               IF (gtyp_SSC.Horizontal_Axis.di_Actual_Position <= (ldi_Pos_Horizontal + gtyp_SSC.Horizontal_Axis.Config.di_Pos_Window))
                   AND (gtyp_SSC.Horizontal_Axis.di_Actual_Position >= (ldi_Pos_Horizontal - gtyp_SSC.Horizontal_Axis.Config.di_Pos_Window))
                   AND gtyp_SSC.Horizontal_Axis.x_Position_Reached
                   AND (gtyp_SSC.Vertical_Axis.di_Actual_Position <= (ldi_Pos_Vertical + gtyp_SSC.Vertical_Axis.Config.di_Pos_Window))
                   AND (gtyp_SSC.Vertical_Axis.di_Actual_Position >= (ldi_Pos_Vertical - gtyp_SSC.Vertical_Axis.Config.di_Pos_Window))
                   AND gtyp_SSC.Vertical_Axis.x_Position_Reached THEN
                   gtyp_SSC.Horizontal_Axis.x_Start_Positioning := FALSE;
                   gtyp_SSC.Vertical_Axis.x_Start_Positioning := FALSE;
                   gtyp_Setup.x_Start_Positioning := FALSE;
                   li_StepCase := 60;
               END_IF;

           60:


               IF gtyp_Setup.x_Start_Positioning OR gtyp_Setup.x_Home_Positioning THEN
                   lx_Start_Positioning_m := TRUE;
                   li_StepCase            := 10;
               ELSIF lfb_R_Trig_Deaktivate.Q THEN
                   gtyp_Setup.x_Home_Positioning := FALSE;
                   li_StepCase                    := 70;
               END_IF;

           70:

               gtyp_SSC.Horizontal_Axis.x_Reference := TRUE;
               gtyp_SSC.Vertical_Axis.x_Reference := TRUE;

               IF NOT gtyp_SSC.Horizontal_Axis.x_Referenced AND NOT gtyp_SSC.Vertical_Axis.x_Referenced THEN
                   li_StepCase := 80;
               END_IF;

           80:
               IF gtyp_SSC.Horizontal_Axis.x_Referenced THEN
                   gtyp_SSC.Horizontal_Axis.x_Reference := FALSE;
               END_IF;
               IF gtyp_SSC.Vertical_Axis.x_Referenced THEN
                   gtyp_SSC.Vertical_Axis.x_Reference := FALSE;
               END_IF;

               IF gtyp_SSC.Horizontal_Axis.x_Referenced AND gtyp_SSC.Vertical_Axis.x_Referenced THEN
                   gtyp_SSC.Horizontal_Axis.x_Reference := FALSE;
                   gtyp_SSC.Vertical_Axis.x_Reference := FALSE;
                   li_StepCase := 0;
               END_IF;


           ELSE
               ;
       END_CASE;

       IF ((gtyp_Setup.i_Pos_Selection > 0)
           AND (gtyp_Setup.i_Pos_Selection < 21)) THEN

           gtyp_Setup.di_Pos_Horizontal := ldi_Pos_Horizontal;
           gtyp_Setup.di_Pos_Vertical := ldi_Pos_Vertical;
           gtyp_Setup.di_Pos_Rotate := 0;
       END_IF;
   ELSE
       lx_Init := TRUE;
   END_IF;
END_FUNCTION_BLOCK

FUNCTION_BLOCK PRG_HBW_Set_Positioning
   VAR
      lx_Init : Bool;
      lx_Start_TON_Wait : Bool;
      lx_Start_Positioning_m : Bool;
      lx_Start_FinalPositioning_m : Bool;
      lx_Start_Offset_m : Bool;
      lt_TON_Wait : Time;
      li_Counter_Hor : Int;
      li_Counter_Ver : Int;
      li_Counter_Act_Hor : Int;
      li_Counter_Act_Ver : Int;
      li_Counter : Int;
      li_StepCase : Int;
      ldi_Pos_Horizontal : DInt;
      ldi_Pos_Vertical : DInt;
      ldi_Offset_Vertical : DInt;
      lfb_R_Trig_Deaktivate : R_TRIG;
      lfb_TON_Wait : TON_TIME;
   END_VAR



   IF lx_Init THEN


       lfb_TON_Wait(IN := lx_Start_TON_Wait,
                     PT := lt_TON_Wait);

       lfb_R_Trig_Deaktivate(CLK:= NOT gtyp_Setup.x_Set_Pos_Activ
                              OR NOT ((gtyp_Setup.i_Pos_Selection > 20)
                              AND (gtyp_Setup.i_Pos_Selection < 41)));

       IF lfb_R_Trig_Deaktivate.Q THEN
           gtyp_HBW.Horizontal_Axis.x_Start_Positioning := FALSE;
           gtyp_HBW.Vertical_Axis.x_Start_Positioning := FALSE;
           gtyp_HBW.Horizontal_Axis.x_Reference := FALSE;
           gtyp_HBW.Vertical_Axis.x_Reference := FALSE;
           gtyp_Setup.x_Start_Positioning := FALSE;
           gtyp_Setup.x_Final_Positioning := FALSE;
           gtyp_Setup.x_Home_Positioning := FALSE;
           gtyp_Setup.x_Start_Offset := FALSE;
           QX_HBW_M4_CantileverBackward_Q8 := FALSE;
           QX_HBW_M4_CantileverForward_Q7 := FALSE;
           IF (li_StepCase > 10) THEN
               li_StepCase := 110;
           END_IF;
       END_IF;


       IF gtyp_Setup.x_Set_Pos_Activ
           AND ((gtyp_Setup.i_Pos_Selection > 20)
           AND (gtyp_Setup.i_Pos_Selection < 41))
           AND ((li_StepCase = 40)
           OR (li_StepCase = 60)
           OR (li_StepCase = 80)
           OR (li_StepCase = 100)) THEN



           IF gtyp_Setup.i_Pos_Selection = 21 THEN
               ldi_Pos_Horizontal := gtyp_HBW.di_PosBelt_Horizontal;
               ldi_Pos_Vertical := gtyp_HBW.di_PosBelt_Vertical;
               ldi_Offset_Vertical := gtyp_HBW.di_Offset_Pos_Belt_Vertical;

           ELSIF gtyp_Setup.i_Pos_Selection = 22 THEN
               ldi_Pos_Horizontal := gtyp_HBW.di_PosRack_A1_Horizontal;
               ldi_Pos_Vertical := gtyp_HBW.di_PosRack_A1_Vertical;
               ldi_Offset_Vertical := gtyp_HBW.di_Offset_Pos_Rack_Vertical;

           ELSIF gtyp_Setup.i_Pos_Selection = 23 THEN
               ldi_Pos_Horizontal := gtyp_HBW.di_PosRack_B2_Horizontal;
               ldi_Pos_Vertical := gtyp_HBW.di_PosRack_B2_Vertical;
               ldi_Offset_Vertical := gtyp_HBW.di_Offset_Pos_Rack_Vertical;

           ELSIF gtyp_Setup.i_Pos_Selection = 24 THEN
               ldi_Pos_Horizontal := gtyp_HBW.di_PosRack_C3_Horizontal;
               ldi_Pos_Vertical := gtyp_HBW.di_PosRack_C3_Vertical;
               ldi_Offset_Vertical := gtyp_HBW.di_Offset_Pos_Rack_Vertical;
           END_IF;
       END_IF;


       IF NOT gtyp_Setup.x_Set_Pos_Activ THEN
           gtyp_Setup.i_Pos_Selection := 0;
       END_IF;


       CASE li_StepCase OF

           0:
               lx_Start_TON_Wait := FALSE;
               li_StepCase := 10;

           10:
               IF gtyp_Setup.x_Set_Pos_Activ
                   AND ((gtyp_Setup.i_Pos_Selection > 20)
                   AND (gtyp_Setup.i_Pos_Selection < 41)) THEN

                   gtyp_HBW.Horizontal_Axis.x_Start_Positioning  := FALSE;
                   gtyp_HBW.Vertical_Axis.x_Start_Positioning    := FALSE;
                   gtyp_HBW.Horizontal_Axis.x_Reference          := FALSE;
                   gtyp_HBW.Vertical_Axis.x_Reference            := FALSE;
                   gtyp_Setup.x_Start_Positioning            := FALSE;
                   gtyp_Setup.x_Final_Positioning            := FALSE;
                   gtyp_Setup.x_Home_Positioning             := FALSE;
                   gtyp_Setup.x_Start_Offset                 := FALSE;
                   QX_HBW_M4_CantileverBackward_Q8               := FALSE;
                   QX_HBW_M4_CantileverForward_Q7                := FALSE;
                   li_StepCase                                    := 20;
               END_IF;

           20:

               gtyp_HBW.Horizontal_Axis.x_Reference := TRUE;
               gtyp_HBW.Vertical_Axis.x_Reference := TRUE;

               IF NOT gtyp_HBW.Horizontal_Axis.x_Referenced AND NOT gtyp_HBW.Vertical_Axis.x_Referenced THEN
                   li_StepCase := 30;
               END_IF;

           30:
               IF gtyp_HBW.Horizontal_Axis.x_Referenced THEN
                   gtyp_HBW.Horizontal_Axis.x_Reference := FALSE;
               END_IF;
               IF gtyp_HBW.Vertical_Axis.x_Referenced THEN
                   gtyp_HBW.Vertical_Axis.x_Reference := FALSE;
               END_IF;

               IF gtyp_HBW.Horizontal_Axis.x_Referenced AND gtyp_HBW.Vertical_Axis.x_Referenced THEN
                   gtyp_HBW.Horizontal_Axis.x_Reference := FALSE;
                   gtyp_HBW.Vertical_Axis.x_Reference := FALSE;
                   li_StepCase := 40;
               END_IF;

           40:
               IF gtyp_Setup.x_Start_Positioning OR lx_Start_Positioning_m OR lx_Start_FinalPositioning_m OR lx_Start_Offset_m THEN
                   lx_Start_Positioning_m := FALSE;
                   li_StepCase := 50;
               END_IF;

           50:
               gtyp_HBW.Horizontal_Axis.di_Target_Position   := ldi_Pos_Horizontal;
               gtyp_HBW.Horizontal_Axis.x_Start_Positioning  := TRUE;
               gtyp_HBW.Vertical_Axis.di_Target_Position     := ldi_Pos_Vertical;
               gtyp_HBW.Vertical_Axis.x_Start_Positioning    := TRUE;

               IF (gtyp_HBW.Horizontal_Axis.di_Actual_Position <= (ldi_Pos_Horizontal + gtyp_HBW.Horizontal_Axis.Config.di_Pos_Window))
                   AND (gtyp_HBW.Horizontal_Axis.di_Actual_Position >= (ldi_Pos_Horizontal - gtyp_HBW.Horizontal_Axis.Config.di_Pos_Window))
                   AND gtyp_HBW.Horizontal_Axis.x_Position_Reached THEN
                   gtyp_HBW.Horizontal_Axis.x_Start_Positioning := FALSE;
               END_IF;

               IF (gtyp_HBW.Vertical_Axis.di_Actual_Position <= (ldi_Pos_Vertical + gtyp_HBW.Vertical_Axis.Config.di_Pos_Window))
                   AND (gtyp_HBW.Vertical_Axis.di_Actual_Position >= (ldi_Pos_Vertical - gtyp_HBW.Vertical_Axis.Config.di_Pos_Window))
                   AND gtyp_HBW.Vertical_Axis.x_Position_Reached THEN
                   gtyp_HBW.Vertical_Axis.x_Start_Positioning := FALSE;
               END_IF;

               IF (gtyp_HBW.Horizontal_Axis.di_Actual_Position <= (ldi_Pos_Horizontal + gtyp_HBW.Horizontal_Axis.Config.di_Pos_Window))
                   AND (gtyp_HBW.Horizontal_Axis.di_Actual_Position >= (ldi_Pos_Horizontal - gtyp_HBW.Horizontal_Axis.Config.di_Pos_Window))
                   AND gtyp_HBW.Horizontal_Axis.x_Position_Reached
                   AND (gtyp_HBW.Vertical_Axis.di_Actual_Position <= (ldi_Pos_Vertical + gtyp_HBW.Vertical_Axis.Config.di_Pos_Window))
                   AND (gtyp_HBW.Vertical_Axis.di_Actual_Position >= (ldi_Pos_Vertical - gtyp_HBW.Vertical_Axis.Config.di_Pos_Window))
                   AND gtyp_HBW.Vertical_Axis.x_Position_Reached THEN
                   gtyp_HBW.Horizontal_Axis.x_Start_Positioning  := FALSE;
                   gtyp_HBW.Vertical_Axis.x_Start_Positioning    := FALSE;
                   gtyp_Setup.x_Start_Positioning          := FALSE;
                   li_StepCase := 60;
               END_IF;

           60:


               IF gtyp_Setup.x_Start_Positioning THEN
                   lx_Start_Positioning_m := TRUE;
                   li_StepCase := 10;

               ELSIF gtyp_Setup.x_Final_Positioning OR lx_Start_FinalPositioning_m OR lx_Start_Offset_m THEN
                   lx_Start_FinalPositioning_m := FALSE;
                   li_StepCase := 70;

               ELSIF lfb_R_Trig_Deaktivate.Q OR gtyp_Setup.x_Home_Positioning THEN
                   gtyp_Setup.x_Home_Positioning := FALSE;
                   li_StepCase := 110;
               END_IF;

           70:

               QX_HBW_M4_CantileverBackward_Q8 := FALSE;
               QX_HBW_M4_CantileverForward_Q7 := TRUE;

               IF IX_HBW_SwitchCantileverFront_I5 AND NOT IX_HBW_SwitchCantileverBack_I6 THEN
                   QX_HBW_M4_CantileverBackward_Q8 := FALSE;
                   QX_HBW_M4_CantileverForward_Q7 := FALSE;
                   gtyp_Setup.x_Final_Positioning := FALSE;
                   li_StepCase := 80;
               END_IF;

           80:


               IF gtyp_Setup.x_Start_Positioning THEN
                   lx_Start_Positioning_m := TRUE;
                   li_StepCase := 110;

               ELSIF gtyp_Setup.x_Final_Positioning THEN
                   lx_Start_FinalPositioning_m := TRUE;
                   li_StepCase := 110;

               ELSIF gtyp_Setup.x_Start_Offset OR lx_Start_Offset_m THEN
                   lx_Start_Offset_m := FALSE;
                   li_StepCase := 90;

               ELSIF lfb_R_Trig_Deaktivate.Q OR gtyp_Setup.x_Home_Positioning THEN
                   gtyp_Setup.x_Home_Positioning := FALSE;
                   li_StepCase := 110;
               END_IF;

           90:
               gtyp_HBW.Vertical_Axis.di_Target_Position := ldi_Pos_Vertical - ldi_Offset_Vertical;
               gtyp_HBW.Vertical_Axis.x_Start_Positioning := TRUE;

               IF (gtyp_HBW.Vertical_Axis.di_Actual_Position <= (ldi_Pos_Vertical - ldi_Offset_Vertical + gtyp_HBW.Vertical_Axis.Config.di_Pos_Window))
                   AND (gtyp_HBW.Vertical_Axis.di_Actual_Position >= (ldi_Pos_Vertical - ldi_Offset_Vertical - gtyp_HBW.Vertical_Axis.Config.di_Pos_Window))
                   AND gtyp_HBW.Vertical_Axis.x_Position_Reached THEN
                   gtyp_HBW.Vertical_Axis.x_Start_Positioning := FALSE;
                   gtyp_Setup.x_Start_Offset            := FALSE;
                   li_StepCase := 100;
               END_IF;

           100:


               IF gtyp_Setup.x_Start_Positioning THEN
                   lx_Start_Positioning_m := TRUE;
                   li_StepCase := 110;

               ELSIF gtyp_Setup.x_Final_Positioning THEN
                   lx_Start_FinalPositioning_m := TRUE;
                   li_StepCase := 110;

               ELSIF gtyp_Setup.x_Start_Offset THEN
                   lx_Start_Offset_m := true;
                   li_StepCase := 110;

               ELSIF lfb_R_Trig_Deaktivate.Q OR gtyp_Setup.x_Home_Positioning THEN
                   gtyp_Setup.x_Home_Positioning := FALSE;
                   li_StepCase := 110;
               END_IF;

           110:
               gtyp_HBW.Vertical_Axis.di_Target_Position := ldi_Pos_Vertical;
               gtyp_HBW.Vertical_Axis.x_Start_Positioning := TRUE;

               IF (gtyp_HBW.Vertical_Axis.di_Actual_Position <= (ldi_Pos_Vertical + gtyp_HBW.Vertical_Axis.Config.di_Pos_Window))
                   AND (gtyp_HBW.Vertical_Axis.di_Actual_Position >= (ldi_Pos_Vertical - gtyp_HBW.Vertical_Axis.Config.di_Pos_Window))
                   AND gtyp_HBW.Vertical_Axis.x_Position_Reached THEN
                   gtyp_HBW.Vertical_Axis.x_Start_Positioning := FALSE;
                   li_StepCase := 120;
               END_IF;

           120:

               QX_HBW_M4_CantileverBackward_Q8 := TRUE;
               QX_HBW_M4_CantileverForward_Q7 := FALSE;

               IF NOT IX_HBW_SwitchCantileverFront_I5 AND IX_HBW_SwitchCantileverBack_I6 THEN
                   QX_HBW_M4_CantileverBackward_Q8 := FALSE;
                   QX_HBW_M4_CantileverForward_Q7 := FALSE;
                   li_StepCase := 130;
               END_IF;

           130:

               gtyp_HBW.Horizontal_Axis.x_Reference := TRUE;
               gtyp_HBW.Vertical_Axis.x_Reference := TRUE;

               IF NOT gtyp_HBW.Horizontal_Axis.x_Referenced AND NOT gtyp_HBW.Vertical_Axis.x_Referenced THEN
                   li_StepCase := 140;
               END_IF;

           140:
               IF gtyp_HBW.Horizontal_Axis.x_Referenced THEN
                   gtyp_HBW.Horizontal_Axis.x_Reference := FALSE;
               END_IF;
               IF gtyp_HBW.Vertical_Axis.x_Referenced THEN
                   gtyp_HBW.Vertical_Axis.x_Reference := FALSE;
               END_IF;

               IF gtyp_HBW.Horizontal_Axis.x_Referenced AND gtyp_HBW.Vertical_Axis.x_Referenced THEN
                   gtyp_HBW.Horizontal_Axis.x_Reference := FALSE;
                   gtyp_HBW.Vertical_Axis.x_Reference := FALSE;
                   li_StepCase := 0;
               END_IF;


       ELSE
           ;
       END_CASE;

       IF ((gtyp_Setup.i_Pos_Selection > 20)
           AND (gtyp_Setup.i_Pos_Selection < 41)) THEN

           gtyp_Setup.di_Pos_Horizontal := ldi_Pos_Horizontal;
           gtyp_Setup.di_Pos_Vertical := ldi_Pos_Vertical;
           gtyp_Setup.di_Pos_Rotate := 0;
       END_IF;
   ELSE
       lx_Init := TRUE;
   END_IF;
END_FUNCTION_BLOCK

FUNCTION_BLOCK PRG_VGR_Set_Positioning
   VAR
      lx_Init : Bool;
      lx_Start_TON_Wait : Bool;
      lx_Start_Positioning_m : Bool;
      lx_Start_FinalPositioning_m : Bool;
      lx_Start_TON_State : Bool;
      lt_TON_Wait : Time;
      ldt_MQTT : Date_And_Time;
      li_Return_LDT : Int;
      li_Lights : Int;
      li_Lights_old : Int;
      lx_State_activ : Bool;
      li_StepCase : Int;
      li_Counter : Int;
      ldi_Pos_SLD_X : DInt;
      ldi_Pos_SLD_Y : DInt;
      ldi_Pos_SLD_Z : DInt;
      ldi_Pos_Horizontal : DInt;
      ldi_Pos_Vertical : DInt;
      ldi_Pos_Rotate : DInt;
      ldi_Offset_Vertical : DInt;
      ls_Color : String;
      ls_Target : String;
      lfb_TON_Wait : TON_TIME;
      lfb_TON_State : TON_TIME;
      lfb_R_Trig_Deaktivate : R_TRIG;
      lfb_R_Trig_NiO : R_TRIG;
   END_VAR



   IF lx_Init THEN


       lfb_TON_Wait(IN := lx_Start_TON_Wait,
                     PT := lt_TON_Wait);

       lfb_R_Trig_Deaktivate(CLK := NOT gtyp_Setup.x_Set_Pos_Activ
                              OR NOT ((gtyp_Setup.i_Pos_Selection > 40)
                              AND (gtyp_Setup.i_Pos_Selection < 61)));

       IF lfb_R_Trig_Deaktivate.Q THEN
           gtyp_VGR.horizontal_Axis.x_Start_Positioning := FALSE;
           gtyp_VGR.vertical_Axis.x_Start_Positioning := FALSE;
           gtyp_VGR.rotate_Axis.x_Start_Positioning := FALSE;
           gtyp_VGR.horizontal_Axis.x_Reference := FALSE;
           gtyp_VGR.vertical_Axis.x_Reference := FALSE;
           gtyp_VGR.rotate_Axis.x_Reference := FALSE;
           gtyp_Setup.x_Start_Positioning := FALSE;
           gtyp_Setup.x_Final_Positioning := FALSE;
           gtyp_Setup.x_Home_Positioning := FALSE;
           gtyp_Setup.x_Start_Offset := FALSE;
           IF (li_StepCase > 10) THEN
               li_StepCase := 150;
           END_IF;
       END_IF;


       IF gtyp_Setup.x_Set_Pos_Activ
           AND ((gtyp_Setup.i_Pos_Selection > 40)
           AND (gtyp_Setup.i_Pos_Selection < 61))
           AND ((li_StepCase = 80)
           OR (li_StepCase = 120)
           OR (li_StepCase = 140)) THEN



           IF gtyp_Setup.i_Pos_Selection = 41 THEN
               ldi_Pos_Horizontal := gtyp_VGR.di_Pos_Color_horizontal;
               ldi_Pos_Vertical := gtyp_VGR.di_Pos_Color_vertical;
               ldi_Pos_Rotate := gtyp_VGR.di_Pos_Color_rotate;
               ldi_Offset_Vertical := gtyp_VGR.di_Offset_Pos_DSI_NFC_vertical;

           ELSIF gtyp_Setup.i_Pos_Selection = 42 THEN
               ldi_Pos_Horizontal := gtyp_VGR.di_Pos_DSI_horizontal;
               ldi_Pos_Vertical := gtyp_VGR.di_Pos_DSI_Collect_vertical;
               ldi_Pos_Rotate := gtyp_VGR.di_Pos_DSI_rotate;
               ldi_Offset_Vertical := gtyp_VGR.di_Offset_Pos_DSI_NFC_vertical;

           ELSIF gtyp_Setup.i_Pos_Selection = 43 THEN
               ldi_Pos_Horizontal := gtyp_VGR.di_Pos_DSI_horizontal;
               ldi_Pos_Vertical := gtyp_VGR.di_Pos_DSI_Discard_vertical;
               ldi_Pos_Rotate := gtyp_VGR.di_Pos_DSI_rotate;
               ldi_Offset_Vertical := gtyp_VGR.di_Offset_Pos_DSI_NFC_vertical;

           ELSIF gtyp_Setup.i_Pos_Selection = 44 THEN
               ldi_Pos_Horizontal := gtyp_VGR.di_Pos_DSO_horizontal;
               ldi_Pos_Vertical := gtyp_VGR.di_Pos_DSO_Collect_vertical;
               ldi_Pos_Rotate := gtyp_VGR.di_Pos_DSO_rotate;
               ldi_Offset_Vertical := gtyp_VGR.di_Offset_Pos_DSO_vertical;

           ELSIF gtyp_Setup.i_Pos_Selection = 45 THEN
               ldi_Pos_Horizontal := gtyp_VGR.di_Pos_DSO_horizontal;
               ldi_Pos_Vertical := gtyp_VGR.di_Pos_DSO_Discard_vertical;
               ldi_Pos_Rotate := gtyp_VGR.di_Pos_DSO_rotate;
               ldi_Offset_Vertical := gtyp_VGR.di_Offset_Pos_DSO_vertical;

           ELSIF gtyp_Setup.i_Pos_Selection = 46 THEN
               ldi_Pos_Horizontal := gtyp_VGR.di_Pos_HBW_horizontal;
               ldi_Pos_Vertical := gtyp_VGR.di_Pos_HBW_Collect_vertical;
               ldi_Pos_Rotate := gtyp_VGR.di_Pos_HBW_rotate;
               ldi_Offset_Vertical := gtyp_VGR.di_Offset_Pos_HBW_vertical;

           ELSIF gtyp_Setup.i_Pos_Selection = 47 THEN
               ldi_Pos_Horizontal := gtyp_VGR.di_Pos_HBW_horizontal;
               ldi_Pos_Vertical := gtyp_VGR.di_Pos_HBW_Discard_vertical;
               ldi_Pos_Rotate := gtyp_VGR.di_Pos_HBW_rotate;
               ldi_Offset_Vertical := gtyp_VGR.di_Offset_Pos_HBW_vertical;

           ELSIF gtyp_Setup.i_Pos_Selection = 48 THEN
               ldi_Pos_Horizontal := gtyp_VGR.di_Pos_MPO_horizontal;
               ldi_Pos_Vertical := gtyp_VGR.di_Pos_MPO_vertical;
               ldi_Pos_Rotate := gtyp_VGR.di_Pos_MPO_rotate;
               ldi_Offset_Vertical := gtyp_VGR.di_Offset_Pos_MPO_vertical;

           ELSIF gtyp_Setup.i_Pos_Selection = 49 THEN
               ldi_Pos_Horizontal := gtyp_VGR.di_Pos_NFC_horizontal;
               ldi_Pos_Vertical := gtyp_VGR.di_Pos_NFC_vertical;
               ldi_Pos_Rotate := gtyp_VGR.di_Pos_NFC_rotate;
               ldi_Offset_Vertical := gtyp_VGR.di_Offset_Pos_DSI_NFC_vertical;

           ELSIF gtyp_Setup.i_Pos_Selection = 50 THEN
               ldi_Pos_Horizontal := gtyp_VGR.di_Pos_NiO_horizontal;
               ldi_Pos_Vertical := gtyp_VGR.di_Pos_NiO_vertical;
               ldi_Pos_Rotate := gtyp_VGR.di_Pos_NiO_rotate;
               ldi_Offset_Vertical := 500;

           ELSIF gtyp_Setup.i_Pos_Selection = 51 THEN
               ldi_Pos_Horizontal := gtyp_VGR.di_Pos_SLD_Blue_horizontal;
               ldi_Pos_Vertical := gtyp_VGR.di_Pos_SLD_Blue_vertical;
               ldi_Pos_Rotate := gtyp_VGR.di_Pos_SLD_Blue_rotate;
               ldi_Offset_Vertical := 500;

           ELSIF gtyp_Setup.i_Pos_Selection = 52 THEN
               ldi_Pos_Horizontal := gtyp_VGR.di_Pos_SLD_Red_horizontal;
               ldi_Pos_Vertical := gtyp_VGR.di_Pos_SLD_Red_vertical;
               ldi_Pos_Rotate := gtyp_VGR.di_Pos_SLD_Red_rotate;
               ldi_Offset_Vertical := 500;

           ELSIF gtyp_Setup.i_Pos_Selection = 53 THEN
               ldi_Pos_Horizontal := gtyp_VGR.di_Pos_SLD_White_horizontal;
               ldi_Pos_Vertical := gtyp_VGR.di_Pos_SLD_White_vertical;
               ldi_Pos_Rotate := gtyp_VGR.di_Pos_SLD_White_rotate;
               ldi_Offset_Vertical := 500;
           END_IF;
       END_IF;


       IF NOT gtyp_Setup.x_Set_Pos_Activ THEN
           gtyp_Setup.i_Pos_Selection := 0;
       END_IF;


       CASE li_StepCase OF

           0:
               lx_Start_TON_Wait := FALSE;
               li_StepCase := 10;

           10:
               IF gtyp_Setup.x_Set_Pos_Activ
                   AND ((gtyp_Setup.i_Pos_Selection > 40)
                   AND (gtyp_Setup.i_Pos_Selection < 61)) THEN

                   gtyp_VGR.horizontal_Axis.x_Start_Positioning := FALSE;
                   gtyp_VGR.vertical_Axis.x_Start_Positioning := FALSE;
                   gtyp_VGR.rotate_Axis.x_Start_Positioning := FALSE;
                   gtyp_VGR.horizontal_Axis.x_Reference := FALSE;
                   gtyp_VGR.vertical_Axis.x_Reference := FALSE;
                   gtyp_VGR.rotate_Axis.x_Reference := FALSE;
                   gtyp_Setup.x_Start_Positioning := FALSE;
                   gtyp_Setup.x_Final_Positioning := FALSE;
                   gtyp_Setup.x_Home_Positioning := FALSE;
                   gtyp_Setup.x_Start_Offset := FALSE;
                   gtyp_VGR.vertical_Axis.i_PWM := 800;
                   li_StepCase := 20;
               END_IF;

           20:
               gtyp_VGR.vertical_Axis.x_Reference := TRUE;

               IF NOT gtyp_VGR.vertical_Axis.x_Referenced THEN
                   li_StepCase := 30;
               END_IF;

           30:
               IF gtyp_VGR.vertical_Axis.x_Referenced THEN
                   gtyp_VGR.vertical_Axis.x_Reference := FALSE;
                   li_StepCase := 40;
               END_IF;

           40:
               gtyp_VGR.horizontal_Axis.x_Reference := TRUE;

               IF NOT gtyp_VGR.horizontal_Axis.x_Referenced THEN
                   li_StepCase := 50;
               END_IF;

           50:
               IF gtyp_VGR.horizontal_Axis.x_Referenced THEN
                   gtyp_VGR.horizontal_Axis.x_Reference := FALSE;
                   li_StepCase := 60;
               END_IF;

           60:
               gtyp_VGR.rotate_Axis.x_Reference := TRUE;

               IF NOT gtyp_VGR.rotate_Axis.x_Referenced THEN
                   li_StepCase := 70;
               END_IF;

           70:
               IF gtyp_VGR.rotate_Axis.x_Referenced THEN
                   gtyp_VGR.rotate_Axis.x_Reference := FALSE;
                   li_StepCase := 80;
               END_IF;

           80:
               IF gtyp_Setup.x_Start_Positioning OR lx_Start_Positioning_m OR lx_Start_FinalPositioning_m THEN
                   lx_Start_Positioning_m := FALSE;
                   li_StepCase := 90;
               END_IF;

           90:
               gtyp_VGR.rotate_Axis.di_Target_Position   := ldi_Pos_Rotate;
               gtyp_VGR.rotate_Axis.x_Start_Positioning  := TRUE;

               IF (gtyp_VGR.rotate_Axis.di_Actual_Position <= (ldi_Pos_Rotate + gtyp_VGR.rotate_Axis.Config.di_Pos_Window))
                   AND (gtyp_VGR.rotate_Axis.di_Actual_Position >= (ldi_Pos_Rotate - gtyp_VGR.rotate_Axis.Config.di_Pos_Window))
                   AND gtyp_VGR.rotate_Axis.x_Position_Reached THEN
                   gtyp_VGR.rotate_Axis.x_Start_Positioning := FALSE;
                   li_StepCase := 100;
               END_IF;

           100:
               gtyp_VGR.horizontal_Axis.di_Target_Position := ldi_Pos_Horizontal;
               gtyp_VGR.horizontal_Axis.x_Start_Positioning := TRUE;

               IF (gtyp_VGR.horizontal_Axis.di_Actual_Position <= (ldi_Pos_Horizontal + gtyp_VGR.horizontal_Axis.Config.di_Pos_Window))
                   AND (gtyp_VGR.horizontal_Axis.di_Actual_Position >= (ldi_Pos_Horizontal - gtyp_VGR.horizontal_Axis.Config.di_Pos_Window))
                   AND gtyp_VGR.horizontal_Axis.x_Position_Reached THEN
                   gtyp_VGR.horizontal_Axis.x_Start_Positioning := FALSE;
                   li_StepCase := 110;
               END_IF;

           110:
               gtyp_VGR.vertical_Axis.i_PWM := 500;
               gtyp_VGR.vertical_Axis.di_Target_Position := ldi_Pos_Vertical - ldi_Offset_Vertical;
               gtyp_VGR.vertical_Axis.x_Start_Positioning := TRUE;

               IF (gtyp_VGR.vertical_Axis.di_Actual_Position <= (ldi_Pos_Vertical - ldi_Offset_Vertical + gtyp_VGR.vertical_Axis.Config.di_Pos_Window))
                   AND (gtyp_VGR.vertical_Axis.di_Actual_Position >= (ldi_Pos_Vertical - ldi_Offset_Vertical - gtyp_VGR.vertical_Axis.Config.di_Pos_Window))
                   AND gtyp_VGR.vertical_Axis.x_Position_Reached THEN
                   gtyp_VGR.vertical_Axis.x_Start_Positioning := FALSE;
                   gtyp_Setup.x_Start_Positioning := FALSE;
                   li_StepCase := 120;
               END_IF;

           120:


               IF gtyp_Setup.x_Start_Positioning THEN
                   lx_Start_Positioning_m := TRUE;
                   li_StepCase := 10;

               ELSIF gtyp_Setup.x_Final_Positioning OR lx_Start_FinalPositioning_m THEN
                   lx_Start_FinalPositioning_m := FALSE;
                   li_StepCase := 130;

               ELSIF lfb_R_Trig_Deaktivate.Q OR gtyp_Setup.x_Home_Positioning THEN
                   gtyp_Setup.x_Home_Positioning := FALSE;
                   li_StepCase := 150;
               END_IF;

           130:
               gtyp_VGR.vertical_Axis.di_Target_Position := ldi_Pos_Vertical;
               gtyp_VGR.vertical_Axis.x_Start_Positioning := TRUE;

               IF (gtyp_VGR.vertical_Axis.di_Actual_Position <= (ldi_Pos_Vertical + gtyp_VGR.vertical_Axis.Config.di_Pos_Window))
                   AND (gtyp_VGR.vertical_Axis.di_Actual_Position >= (ldi_Pos_Vertical - gtyp_VGR.vertical_Axis.Config.di_Pos_Window))
                   AND gtyp_VGR.vertical_Axis.x_Position_Reached THEN
                   gtyp_VGR.vertical_Axis.x_Start_Positioning := FALSE;
                   gtyp_Setup.x_Final_Positioning := FALSE;
                   li_StepCase := 140;
               END_IF;

           140:


               IF gtyp_Setup.x_Start_Positioning THEN
                   lx_Start_Positioning_m := TRUE;
                   li_StepCase := 10;

               ELSIF gtyp_Setup.x_Final_Positioning THEN
                   lx_Start_FinalPositioning_m := TRUE;
                   li_StepCase := 10;

               ELSIF lfb_R_Trig_Deaktivate.Q OR gtyp_Setup.x_Home_Positioning THEN
                   gtyp_Setup.x_Home_Positioning := FALSE;
                   li_StepCase := 150;
               END_IF;

           150:
               gtyp_VGR.vertical_Axis.i_PWM := 800;
               gtyp_VGR.vertical_Axis.x_Reference := TRUE;

               IF NOT gtyp_VGR.vertical_Axis.x_Referenced THEN
                   li_StepCase := 160;
               END_IF;

           160:
               IF gtyp_VGR.vertical_Axis.x_Referenced THEN
                   gtyp_VGR.vertical_Axis.x_Reference := FALSE;
                   li_StepCase := 170;
               END_IF;

           170:
               gtyp_VGR.horizontal_Axis.x_Reference := TRUE;

               IF NOT gtyp_VGR.horizontal_Axis.x_Referenced THEN
                   li_StepCase := 180;
               END_IF;

           180:
               IF gtyp_VGR.horizontal_Axis.x_Referenced THEN
                   gtyp_VGR.horizontal_Axis.x_Reference := FALSE;
                   li_StepCase := 0;
               END_IF;


           ELSE
               ;
       END_CASE;

       IF ((gtyp_Setup.i_Pos_Selection > 40)
           AND (gtyp_Setup.i_Pos_Selection < 61)) THEN

           gtyp_Setup.di_Pos_Horizontal := ldi_Pos_Horizontal;
           gtyp_Setup.di_Pos_Vertical := ldi_Pos_Vertical;
           gtyp_Setup.di_Pos_Rotate := ldi_Pos_Rotate;
       END_IF;
   ELSE
       lx_Init := TRUE;
   END_IF;
END_FUNCTION_BLOCK

FUNCTION_BLOCK PRG_SSC_Ablauf
   VAR
      lx_Init : Bool;
      lx_FirstCentre : Bool;
      lx_Start : Bool;
      lx_Start_TON_State : Bool;
      lt_TON_Wait : Time;
      li_StepCase : Int;
      ldi_TargetPosition_Horizontal : DInt;
      ldi_TargetPosition_Vertical : DInt;
      lldt_ts_old : LDT;
      ldt_write : Date_And_Time;
      li_Return_write : Int;
      ldt_MQTT : Date_And_Time;
      li_Return_LDT : Int;
      lx_Start_TON_Wait : Bool;
      ldi_StepHorizontal : DInt;
      ldi_StepVertical : DInt;
      lfb_TON_Wait : TON_TIME;
      lfb_TON_State : TON_TIME;
      lfb_F_TRIG_Set_Pos : F_TRIG;
   END_VAR



   IF lx_Init THEN


       IF gtyp_Setup.x_Set_Pos_Activ OR gtyp_SSC.x_Start_Park_Position THEN
           li_StepCase := 0;
       END_IF;


       lfb_F_TRIG_Set_Pos(CLK:= gtyp_Setup.x_Set_Pos_Activ);

       IF lfb_F_TRIG_Set_Pos.Q THEN
           lx_FirstCentre := TRUE;
       END_IF;

       lfb_TON_Wait(IN := lx_Start_TON_Wait,
                        PT := lt_TON_Wait);


       lfb_TON_State(IN := NOT lx_Start_TON_State,
                      PT := T#2s);


       IF lfb_TON_State.Q AND NOT lx_Start_TON_State THEN
           lx_Start_TON_State := TRUE;
           li_Return_LDT := RD_SYS_T(ldt_MQTT);
           gtyp_Interface_Dashboard.Subscribe.PosPanTiltUnit.ldt_ts := DT_TO_LDT(ldt_MQTT);
       END_IF;


       IF NOT lfb_TON_State.Q AND lx_Start_TON_State THEN
           lx_Start_TON_State := FALSE;
       END_IF;

       CASE li_StepCase OF

           0:
               lx_Start_TON_State := FALSE;
               gtyp_SSC.Horizontal_Axis.x_Start_Positioning  := FALSE;
               gtyp_SSC.Vertical_Axis.x_Start_Positioning    := FALSE;

               IF NOT gtyp_Setup.x_Set_Pos_Activ AND NOT gtyp_SSC.x_Start_Park_Position THEN
                   li_StepCase := 10;
               END_IF;

           10:

               IF (gtyp_Interface_Dashboard.Publish.PosPanTiltUnit.ldt_ts > lldt_ts_old) OR lx_FirstCentre THEN

                   lldt_ts_old := gtyp_Interface_Dashboard.Publish.PosPanTiltUnit.ldt_ts;


                   ldi_StepHorizontal := REAL_TO_DINT(FC_Scale_linear(inr_Y1 := DINT_TO_REAL(gtyp_SSC.Horizontal_Axis.Config.di_Neg_Soft_Switch),
                                                                                                             inr_Y2 := DINT_TO_REAL(gtyp_SSC.Horizontal_Axis.Config.di_Pos_Soft_Switch),
                                                                                                             inr_X1 := 0.0,
                                                                                                             inr_X2 := 180.0,
                                                                                                             inr_X := DINT_TO_REAL(gtyp_Interface_Dashboard.Publish.PosPanTiltUnit.i_degree)));
                   ldi_StepVertical := REAL_TO_DINT(FC_Scale_linear(inr_Y1 := DINT_TO_REAL(gtyp_SSC.Vertical_Axis.Config.di_Neg_Soft_Switch),
                                                                                                         inr_Y2 := DINT_TO_REAL(gtyp_SSC.Vertical_Axis.Config.di_Pos_Soft_Switch),
                                                                                                         inr_X1 := 0.0,
                                                                                                         inr_X2 := 180.0,
                                                                                                         inr_X := DINT_TO_REAL(gtyp_Interface_Dashboard.Publish.PosPanTiltUnit.i_degree)));

                   IF (gtyp_Interface_Dashboard.Publish.PosPanTiltUnit.s_cmd = 'relmove_left')
                       AND ((gtyp_SSC.Horizontal_Axis.di_Actual_Position - ldi_StepHorizontal) > gtyp_SSC.Horizontal_Axis.Config.di_Neg_Soft_Switch + 15)
                       AND NOT IX_SSC_RefSwitchHorizontalAxis_I2 THEN
                       ldi_TargetPosition_Horizontal := gtyp_SSC.Horizontal_Axis.di_Actual_Position - ldi_StepHorizontal;
                       gtyp_SSC.Horizontal_Axis.di_Target_Position := ldi_TargetPosition_Horizontal;
                       gtyp_SSC.Horizontal_Axis.x_Start_Positioning := TRUE;
                       li_StepCase := 70;

                   ELSIF (gtyp_Interface_Dashboard.Publish.PosPanTiltUnit.s_cmd = 'relmove_right')
                       AND ((gtyp_SSC.Horizontal_Axis.di_Actual_Position + ldi_StepHorizontal) < gtyp_SSC.Horizontal_Axis.Config.di_Pos_Soft_Switch - 15) THEN
                       ldi_TargetPosition_Horizontal := gtyp_SSC.Horizontal_Axis.di_Actual_Position + ldi_StepHorizontal;
                       gtyp_SSC.Horizontal_Axis.di_Target_Position := ldi_TargetPosition_Horizontal;
                       gtyp_SSC.Horizontal_Axis.x_Start_Positioning := TRUE;
                       li_StepCase := 70;

                   ELSIF (gtyp_Interface_Dashboard.Publish.PosPanTiltUnit.s_cmd = 'relmove_up')
                       AND ((gtyp_SSC.Vertical_Axis.di_Actual_Position + ldi_StepHorizontal) < gtyp_SSC.Vertical_Axis.Config.di_Pos_Soft_Switch - 15) THEN
                       ldi_TargetPosition_Vertical := gtyp_SSC.Vertical_Axis.di_Actual_Position + ldi_StepVertical;
                       gtyp_SSC.Vertical_Axis.di_Target_Position := ldi_TargetPosition_Vertical;
                       gtyp_SSC.Vertical_Axis.x_Start_Positioning := TRUE;
                       li_StepCase := 80;

                   ELSIF (gtyp_Interface_Dashboard.Publish.PosPanTiltUnit.s_cmd = 'relmove_down')
                       AND ((gtyp_SSC.Vertical_Axis.di_Actual_Position - ldi_StepVertical) > gtyp_SSC.Vertical_Axis.Config.di_Neg_Soft_Switch + 15)
                       AND NOT IX_SSC_RefSwitchVerticalAxis_I1 THEN
                       ldi_TargetPosition_Vertical := gtyp_SSC.Vertical_Axis.di_Actual_Position - ldi_StepVertical;
                       gtyp_SSC.Vertical_Axis.di_Target_Position := ldi_TargetPosition_Vertical;
                       gtyp_SSC.Vertical_Axis.x_Start_Positioning := TRUE;
                       li_StepCase := 80;

                   ELSIF lx_FirstCentre THEN
                       li_StepCase := 20;

                   ELSIF (gtyp_Interface_Dashboard.Publish.PosPanTiltUnit.s_cmd = 'home') THEN
                       li_StepCase := 60;

                   ELSIF (gtyp_Interface_Dashboard.Publish.PosPanTiltUnit.s_cmd = 'start_pan')
                       AND (gtyp_SSC.Horizontal_Axis.di_Actual_Position > gtyp_SSC.Horizontal_Axis.Config.di_Neg_Soft_Switch + 15)
                       AND NOT IX_SSC_RefSwitchHorizontalAxis_I2 THEN
                       ldi_TargetPosition_Horizontal := gtyp_SSC.Horizontal_Axis.Config.di_Neg_Soft_Switch + 15;
                       gtyp_SSC.Horizontal_Axis.di_Target_Position := ldi_TargetPosition_Horizontal;
                       gtyp_SSC.Horizontal_Axis.x_Start_Positioning := TRUE;
                       li_StepCase := 70;

                   ELSIF (gtyp_Interface_Dashboard.Publish.PosPanTiltUnit.s_cmd = 'end_pan')
                       AND (gtyp_SSC.Horizontal_Axis.di_Actual_Position < gtyp_SSC.Horizontal_Axis.Config.di_Pos_Soft_Switch - 15) THEN
                       ldi_TargetPosition_Horizontal := gtyp_SSC.Horizontal_Axis.Config.di_Pos_Soft_Switch - 15;
                       gtyp_SSC.Horizontal_Axis.di_Target_Position := ldi_TargetPosition_Horizontal;
                       gtyp_SSC.Horizontal_Axis.x_Start_Positioning := TRUE;
                       li_StepCase := 70;

                   ELSIF (gtyp_Interface_Dashboard.Publish.PosPanTiltUnit.s_cmd = 'start_tilt')
                       AND (gtyp_SSC.Vertical_Axis.di_Actual_Position > gtyp_SSC.Vertical_Axis.Config.di_Neg_Soft_Switch + 15)
                       AND NOT IX_SSC_RefSwitchVerticalAxis_I1 THEN
                       ldi_TargetPosition_Vertical := gtyp_SSC.Vertical_Axis.Config.di_Neg_Soft_Switch + 15;
                       gtyp_SSC.Vertical_Axis.di_Target_Position := ldi_TargetPosition_Vertical;
                       gtyp_SSC.Vertical_Axis.x_Start_Positioning := TRUE;
                       li_StepCase := 80;

                   ELSIF (gtyp_Interface_Dashboard.Publish.PosPanTiltUnit.s_cmd = 'end_tilt')
                       AND (gtyp_SSC.Vertical_Axis.di_Actual_Position < gtyp_SSC.Vertical_Axis.Config.di_Pos_Soft_Switch - 15) THEN
                       ldi_TargetPosition_Vertical := gtyp_SSC.Vertical_Axis.Config.di_Pos_Soft_Switch - 15;
                       gtyp_SSC.Vertical_Axis.di_Target_Position := ldi_TargetPosition_Vertical;
                       gtyp_SSC.Vertical_Axis.x_Start_Positioning := TRUE;
                       li_StepCase := 80;
                   END_IF;
               END_IF;

           20:
               gtyp_SSC.Horizontal_Axis.x_Reference  := TRUE;
               gtyp_SSC.Vertical_Axis.x_Reference    := TRUE;

               IF NOT gtyp_SSC.Horizontal_Axis.x_Referenced AND NOT gtyp_SSC.Vertical_Axis.x_Referenced THEN
                  li_StepCase := 30;
               END_IF;

           30:
               IF gtyp_SSC.Horizontal_Axis.x_Referenced THEN
                   gtyp_SSC.Horizontal_Axis.x_Reference := FALSE;
               END_IF;
               IF gtyp_SSC.Vertical_Axis.x_Referenced THEN
                   gtyp_SSC.Vertical_Axis.x_Reference := FALSE;
               END_IF;

               IF gtyp_SSC.Horizontal_Axis.x_Referenced AND gtyp_SSC.Vertical_Axis.x_Referenced THEN
                   gtyp_SSC.Horizontal_Axis.x_Reference := FALSE;
                   gtyp_SSC.Vertical_Axis.x_Reference := FALSE;
                   lx_Start_TON_Wait := TRUE;
                   li_StepCase := 40;
               END_IF;

           40:
               IF lfb_TON_Wait.Q THEN
                   lx_Start_TON_Wait := FALSE;
                   li_StepCase := 50;
               END_IF;

           50:
               gtyp_SSC.Horizontal_Axis.di_Target_Position   := gtyp_SSC.di_Pos_HBW_Horizontal;
               gtyp_SSC.Horizontal_Axis.x_Start_Positioning  := TRUE;
               gtyp_SSC.Vertical_Axis.di_Target_Position     := gtyp_SSC.di_Pos_HBW_Vertical;
               gtyp_SSC.Vertical_Axis.x_Start_Positioning    := TRUE;

               IF (gtyp_SSC.Horizontal_Axis.di_Actual_Position <= (gtyp_SSC.di_Pos_HBW_Horizontal + gtyp_SSC.Horizontal_Axis.Config.di_Pos_Window))
                   AND (gtyp_SSC.Horizontal_Axis.di_Actual_Position >= (gtyp_SSC.di_Pos_HBW_Horizontal - gtyp_SSC.Horizontal_Axis.Config.di_Pos_Window))
                   AND gtyp_SSC.Horizontal_Axis.x_Position_Reached THEN
                   gtyp_SSC.Horizontal_Axis.x_Start_Positioning := FALSE;
               END_IF;

               IF (gtyp_SSC.Vertical_Axis.di_Actual_Position <= (gtyp_SSC.di_Pos_HBW_Vertical + gtyp_SSC.Vertical_Axis.Config.di_Pos_Window))
                   AND (gtyp_SSC.Vertical_Axis.di_Actual_Position >= (gtyp_SSC.di_Pos_HBW_Vertical - gtyp_SSC.Vertical_Axis.Config.di_Pos_Window))
                   AND gtyp_SSC.Vertical_Axis.x_Position_Reached THEN
                   gtyp_SSC.Vertical_Axis.x_Start_Positioning := FALSE;
               END_IF;

               IF (gtyp_SSC.Horizontal_Axis.di_Actual_Position <= (gtyp_SSC.di_Pos_HBW_Horizontal + gtyp_SSC.Horizontal_Axis.Config.di_Pos_Window))
                   AND (gtyp_SSC.Horizontal_Axis.di_Actual_Position >= (gtyp_SSC.di_Pos_HBW_Horizontal - gtyp_SSC.Horizontal_Axis.Config.di_Pos_Window))
                   AND gtyp_SSC.Horizontal_Axis.x_Position_Reached
                   AND (gtyp_SSC.Vertical_Axis.di_Actual_Position <= (gtyp_SSC.di_Pos_HBW_Vertical + gtyp_SSC.Vertical_Axis.Config.di_Pos_Window))
                   AND (gtyp_SSC.Vertical_Axis.di_Actual_Position >= (gtyp_SSC.di_Pos_HBW_Vertical - gtyp_SSC.Vertical_Axis.Config.di_Pos_Window))
                   AND gtyp_SSC.Vertical_Axis.x_Position_Reached THEN
                   gtyp_SSC.Horizontal_Axis.x_Start_Positioning := FALSE;
                   gtyp_SSC.Vertical_Axis.x_Start_Positioning := FALSE;
                   lx_FirstCentre := FALSE;
                   li_StepCase := 90;
               END_IF;

           60:
               gtyp_SSC.Horizontal_Axis.di_Target_Position := gtyp_SSC.di_Pos_Centre_Horizontal;
               gtyp_SSC.Horizontal_Axis.x_Start_Positioning := TRUE;
               gtyp_SSC.Vertical_Axis.di_Target_Position := gtyp_SSC.di_Pos_Centre_Vertical;
               gtyp_SSC.Vertical_Axis.x_Start_Positioning := TRUE;

               IF (gtyp_SSC.Horizontal_Axis.di_Actual_Position <= (gtyp_SSC.di_Pos_Centre_Horizontal + gtyp_SSC.Horizontal_Axis.Config.di_Pos_Window))
                   AND (gtyp_SSC.Horizontal_Axis.di_Actual_Position >= (gtyp_SSC.di_Pos_Centre_Horizontal - gtyp_SSC.Horizontal_Axis.Config.di_Pos_Window))
                   AND gtyp_SSC.Horizontal_Axis.x_Position_Reached THEN
                   gtyp_SSC.Horizontal_Axis.x_Start_Positioning := FALSE;
               END_IF;

               IF (gtyp_SSC.Vertical_Axis.di_Actual_Position <= (gtyp_SSC.di_Pos_Centre_Vertical + gtyp_SSC.Vertical_Axis.Config.di_Pos_Window))
                   AND (gtyp_SSC.Vertical_Axis.di_Actual_Position >= (gtyp_SSC.di_Pos_Centre_Vertical - gtyp_SSC.Vertical_Axis.Config.di_Pos_Window))
                   AND gtyp_SSC.Vertical_Axis.x_Position_Reached THEN
                   gtyp_SSC.Vertical_Axis.x_Start_Positioning := FALSE;
               END_IF;

               IF (gtyp_SSC.Horizontal_Axis.di_Actual_Position <= (gtyp_SSC.di_Pos_Centre_Horizontal + gtyp_SSC.Horizontal_Axis.Config.di_Pos_Window))
                   AND (gtyp_SSC.Horizontal_Axis.di_Actual_Position >= (gtyp_SSC.di_Pos_Centre_Horizontal - gtyp_SSC.Horizontal_Axis.Config.di_Pos_Window))
                   AND gtyp_SSC.Horizontal_Axis.x_Position_Reached
                   AND (gtyp_SSC.Vertical_Axis.di_Actual_Position <= (gtyp_SSC.di_Pos_Centre_Vertical + gtyp_SSC.Vertical_Axis.Config.di_Pos_Window))
                   AND (gtyp_SSC.Vertical_Axis.di_Actual_Position >= (gtyp_SSC.di_Pos_Centre_Vertical - gtyp_SSC.Vertical_Axis.Config.di_Pos_Window))
                   AND gtyp_SSC.Vertical_Axis.x_Position_Reached THEN
                   gtyp_SSC.Horizontal_Axis.x_Start_Positioning := FALSE;
                   gtyp_SSC.Vertical_Axis.x_Start_Positioning := FALSE;
                   lx_FirstCentre := FALSE;
                   li_StepCase := 90;
               END_IF;

           70:
               IF (gtyp_SSC.Horizontal_Axis.di_Actual_Position <= (ldi_TargetPosition_Horizontal + gtyp_SSC.Horizontal_Axis.Config.di_Pos_Window))
                   AND (gtyp_SSC.Horizontal_Axis.di_Actual_Position >= (ldi_TargetPosition_Horizontal - gtyp_SSC.Horizontal_Axis.Config.di_Pos_Window))
                   AND gtyp_SSC.Horizontal_Axis.x_Position_Reached THEN
                   gtyp_SSC.Horizontal_Axis.x_Start_Positioning := FALSE;
                   li_StepCase := 90;
               END_IF;

           80:
               IF (gtyp_SSC.Vertical_Axis.di_Actual_Position <= (ldi_TargetPosition_Vertical + gtyp_SSC.Vertical_Axis.Config.di_Pos_Window))
                   AND (gtyp_SSC.Vertical_Axis.di_Actual_Position >= (ldi_TargetPosition_Vertical - gtyp_SSC.Vertical_Axis.Config.di_Pos_Window))
                   AND gtyp_SSC.Vertical_Axis.x_Position_Reached THEN
                   gtyp_SSC.Vertical_Axis.x_Start_Positioning := FALSE;
                   li_StepCase := 90;
               END_IF;

           90:
               gtyp_Interface_Dashboard.Subscribe.PosPanTiltUnit.r_pan := FC_Scale_linear(inr_Y1 := -1.0,
                                                                                              inr_Y2 := 1.0,
                                                                                              inr_X1 := DINT_TO_REAL(gtyp_SSC.Horizontal_Axis.Config.di_Neg_Soft_Switch),
                                                                                              inr_X2 := DINT_TO_REAL(gtyp_SSC.Horizontal_Axis.Config.di_Pos_Soft_Switch),
                                                                                              inr_X := gtyp_SSC.Horizontal_Axis.di_Actual_Position);
               gtyp_Interface_Dashboard.Subscribe.PosPanTiltUnit.r_tilt:= FC_Scale_linear(inr_Y1 := -1.0,
                                                                                              inr_Y2 := 1.0,
                                                                                              inr_X1 := DINT_TO_REAL(gtyp_SSC.Vertical_Axis.Config.di_Neg_Soft_Switch),
                                                                                              inr_X2 := DINT_TO_REAL(gtyp_SSC.Vertical_Axis.Config.di_Pos_Soft_Switch),
                                                                                              inr_X := gtyp_SSC.Vertical_Axis.di_Actual_Position);

               li_Return_write := RD_SYS_T(ldt_write);
               gtyp_Interface_Dashboard.Subscribe.PosPanTiltUnit.ldt_ts := DT_TO_LDT(ldt_write);
               lx_Start_TON_Wait := TRUE;
               li_StepCase := 100;

           100:
               IF lfb_TON_Wait.Q THEN
                   lx_Start_TON_Wait := FALSE;
                   li_StepCase := 0;
               END_IF;

       ELSE
           ;
       END_CASE;

   ELSE
       lx_Init := TRUE;
       lx_FirstCentre := TRUE;

       gtyp_SSC.x_Start_Park_Position := FALSE;
       gtyp_SSC.x_Park_Position_Reached := FALSE;
       gtyp_SSC.x_Error := FALSE;
   END_IF;
END_FUNCTION_BLOCK

FUNCTION_BLOCK PRG_SLD_Calibration_Color
   VAR
      lx_Init : Bool;
      lx_Start_TON_Wait : Bool;
      lx_Start_Positioning_m : Bool;
      lt_TON_Wait : Time;
      li_StepCase : Int;
      lw_ColorValueMin : Word;
      ldi_Pos_Horizontal : DInt;
      ldi_Pos_Vertical : DInt;
      lfb_R_Trig_Deaktivate : R_TRIG;
      lfb_TON_Wait : TON_TIME;
   END_VAR



   IF lx_Init THEN


       lfb_TON_Wait(IN := lx_Start_TON_Wait,
                     PT := lt_TON_Wait);

       lfb_R_Trig_Deaktivate(CLK:= NOT gtyp_Setup.x_Color_Sensor_Calibration
                              OR NOT (gtyp_Setup.i_Color_Sensor_Selection = 2));

       IF lfb_R_Trig_Deaktivate.Q THEN
           gtyp_Setup.x_Calculate_Value_Color := FALSE;
           gtyp_Setup.x_Set_Calib_Value_Color_Blue := FALSE;
           gtyp_Setup.x_Set_Calib_Value_Color_Red := FALSE;
           gtyp_Setup.x_Set_Calib_Value_Color_White := FALSE;
           gtyp_Setup.w_Calib_ColorValue_Blue := 0;
           gtyp_Setup.w_Calib_ColorValue_Red := 0;
           gtyp_Setup.w_Calib_ColorValue_White := 0;
           gtyp_Setup.w_Threshold_Red_Blue := 0;
           gtyp_Setup.w_Threshold_White_Red := 0;
           QX_SLD_M1_ConveyorBelt_Q1 := FALSE;
           lw_ColorValueMin := 16#FF;
           li_StepCase            := 0;
       END_IF;


       CASE li_StepCase OF

           0:
               lx_Start_TON_Wait := FALSE;
               li_StepCase := 10;

           10:
               IF gtyp_Setup.x_Color_Sensor_Calibration
                   AND (gtyp_Setup.i_Color_Sensor_Selection = 2) THEN
                   gtyp_Setup.x_Calculate_Value_Color := FALSE;
                   gtyp_Setup.x_Set_Calib_Value_Color_Blue := FALSE;
                   gtyp_Setup.x_Set_Calib_Value_Color_Red := FALSE;
                   gtyp_Setup.x_Set_Calib_Value_Color_White := FALSE;
                   gtyp_Setup.w_Calib_ColorValue_Blue := 0;
                   gtyp_Setup.w_Calib_ColorValue_Red := 0;
                   gtyp_Setup.w_Calib_ColorValue_White := 0;
                   gtyp_Setup.w_Threshold_Red_Blue := 0;
                   gtyp_Setup.w_Threshold_White_Red := 0;
                   QX_SLD_M1_ConveyorBelt_Q1 := FALSE;
                   lw_ColorValueMin := 16#FFFF;
                   li_StepCase := 20;
               END_IF;

           20:

               IF NOT IX_SLD_LightBarrierInlet_I2 THEN
                   QX_SLD_M1_ConveyorBelt_Q1 := TRUE;
                   lw_ColorValueMin := 16#FFFF;
               END_IF;

               IF lw_ColorValueMin > IW_SLD_ColorSensor_A4 THEN
                   lw_ColorValueMin := IW_SLD_ColorSensor_A4;
               END_IF;

               IF NOT IX_SLD_LightBarrierBehindColorSensor_I3 THEN
                   QX_SLD_M1_ConveyorBelt_Q1 := FALSE;
               END_IF;


               IF gtyp_Setup.x_Set_Calib_Value_Color_Blue THEN
                   gtyp_Setup.w_Calib_ColorValue_Blue := lw_ColorValueMin;
                   gtyp_Setup.x_Set_Calib_Value_Color_Blue := FALSE;
               ELSIF gtyp_Setup.x_Set_Calib_Value_Color_Red THEN
                   gtyp_Setup.w_Calib_ColorValue_Red := lw_ColorValueMin;
                   gtyp_Setup.x_Set_Calib_Value_Color_Red := FALSE;
               ELSIF gtyp_Setup.x_Set_Calib_Value_Color_White THEN
                   gtyp_Setup.w_Calib_ColorValue_White := lw_ColorValueMin;
                   gtyp_Setup.x_Set_Calib_Value_Color_White := FALSE;
               END_IF;

               gtyp_Setup.w_Threshold_White_Red := gtyp_Setup.w_Calib_ColorValue_White + ((gtyp_Setup.w_Calib_ColorValue_Red - gtyp_Setup.w_Calib_ColorValue_White) / 2);
               gtyp_Setup.w_Threshold_Red_Blue := gtyp_Setup.w_Calib_ColorValue_Red + ((gtyp_Setup.w_Calib_ColorValue_Blue - gtyp_Setup.w_Calib_ColorValue_Red) / 2);

               IF gtyp_Setup.x_Calculate_Value_Color THEN
                   gtyp_SLD.w_Threshold_White_Red := gtyp_Setup.w_Threshold_White_Red;
                   gtyp_SLD.w_Threshold_Red_Blue := gtyp_Setup.w_Threshold_Red_Blue;
                   gtyp_Setup.x_Calculate_Value_Color := FALSE;
               END_IF;


           ELSE
               ;
       END_CASE;

       IF (gtyp_Setup.i_Color_Sensor_Selection = 2) THEN

           gtyp_Setup.w_Actual_ColorValue := IW_SLD_ColorSensor_A4;
       END_IF;
   ELSE
       lx_Init := TRUE;
   END_IF;
END_FUNCTION_BLOCK

FUNCTION_BLOCK PRG_SSC_Axis_Vertical
   VAR
      lx_Init : Bool;
      lfb_Vertical_Axis : FB_Axis;
   END_VAR



   IF lx_Init THEN


       lfb_Vertical_Axis( ini_Axis                := 5,
                           indi_Increment          := gtyp_SSC.Vertical_Axis.di_Increment,
                           inx_Ref_Switch          := IX_SSC_RefSwitchVerticalAxis_I1,
                           inx_Referencing         := gtyp_SSC.Vertical_Axis.x_Reference,
                           inx_Start_Positioning   := gtyp_SSC.Vertical_Axis.x_Start_Positioning,
                           indi_Target_Position    := gtyp_SSC.Vertical_Axis.di_Target_Position,
                           ini_PWM               := gtyp_SSC.Vertical_Axis.i_PWM,
                           inouttyp_Config         := gtyp_SSC.Vertical_Axis.Config,
                           inouttyp_Setup          := gtyp_SetupAxis);

       QX_SSC_M1_VerticalAxisUp_Q1                    := lfb_Vertical_Axis.outx_Motor_Pos;
       QX_SSC_M1_VerticalAxisDown_Q2                  := lfb_Vertical_Axis.outx_Motor_Neg;
       QW_SSC_PWM_Vertical_M1                         := lfb_Vertical_Axis.outi_Motor_PWM;
       gtyp_SSC.Vertical_Axis.di_Actual_Position   := lfb_Vertical_Axis.outdi_Actual_Position;
       gtyp_SSC.Vertical_Axis.x_Referenced         := lfb_Vertical_Axis.outx_Referenced;
       gtyp_SSC.Vertical_Axis.x_Position_Reached   := lfb_Vertical_Axis.outx_Position_Reached;
   ELSE
       lx_Init := TRUE;
   END_IF;
END_FUNCTION_BLOCK

FUNCTION_BLOCK PRG_SSC_Set_Park_Position
   VAR
      lx_Init : Bool;
      lx_Start_TON_Wait : Bool;
      lt_TON_Wait : Time;
      li_StepCase : Int;
      lfb_TON_Wait : TON_TIME;
      lfb_R_Trig_Start_Park_Pos : R_TRIG;
   END_VAR



   IF lx_Init THEN


       lfb_TON_Wait(IN := lx_Start_TON_Wait,
                     PT := lt_TON_Wait);

       lfb_R_Trig_Start_Park_Pos(CLK := gtyp_Setup.x_Park_Position
                                  OR IX_Set_Park_Position);


       IF lfb_R_Trig_Start_Park_Pos.Q THEN
           gtyp_SSC.x_Start_Park_Position := TRUE;
           li_StepCase := 0;
       END_IF;


       IF NOT gtyp_SSC.x_Start_Park_Position THEN
           li_StepCase := 0;
       END_IF;


       CASE li_StepCase OF

           0:
               lx_Start_TON_Wait := FALSE;
               li_StepCase := 10;

           10:
               IF gtyp_SSC.x_Start_Park_Position AND NOT gtyp_SSC.x_Park_Position_Reached THEN
                   gtyp_SSC.Horizontal_Axis.x_Start_Positioning := FALSE;
                   gtyp_SSC.Vertical_Axis.x_Start_Positioning := FALSE;
                   gtyp_SSC.Horizontal_Axis.x_Reference := FALSE;
                   gtyp_SSC.Vertical_Axis.x_Reference := FALSE;
                    li_StepCase := 20;
               END_IF;

           20:
               gtyp_SSC.Vertical_Axis.x_Reference := TRUE;

               IF NOT gtyp_SSC.Vertical_Axis.x_Referenced THEN
                   li_StepCase := 30;
               END_IF;

           30:
               IF gtyp_SSC.Vertical_Axis.x_Referenced THEN
                   gtyp_SSC.Vertical_Axis.x_Reference := FALSE;
                   li_StepCase := 40;
               END_IF;

           40:
               gtyp_SSC.Horizontal_Axis.x_Reference := TRUE;

               IF NOT gtyp_SSC.Horizontal_Axis.x_Referenced THEN
                   li_StepCase := 50;
               END_IF;

           50:
               IF gtyp_SSC.Horizontal_Axis.x_Referenced THEN
                   gtyp_SSC.Horizontal_Axis.x_Reference := FALSE;
                   li_StepCase := 60;
               END_IF;

           60:
               gtyp_SSC.Horizontal_Axis.di_Target_Position := gtyp_SSC.di_Pos_Park_Horizontal;
               gtyp_SSC.Horizontal_Axis.x_Start_Positioning := TRUE;

               IF (gtyp_SSC.Horizontal_Axis.di_Actual_Position <= (gtyp_SSC.di_Pos_Park_Horizontal + gtyp_SSC.Horizontal_Axis.Config.di_Pos_Window))
                   AND (gtyp_SSC.Horizontal_Axis.di_Actual_Position >= (gtyp_SSC.di_Pos_Park_Horizontal - gtyp_SSC.Horizontal_Axis.Config.di_Pos_Window))
                   AND gtyp_SSC.Horizontal_Axis.x_Position_Reached THEN
                   gtyp_SSC.Horizontal_Axis.x_Start_Positioning := FALSE;
                   li_StepCase := 70;
               END_IF;

           70:
               gtyp_SSC.Vertical_Axis.di_Target_Position := gtyp_SSC.di_Pos_Park_Vertical;
               gtyp_SSC.Vertical_Axis.x_Start_Positioning := TRUE;

               IF (gtyp_SSC.Vertical_Axis.di_Actual_Position <= (gtyp_SSC.di_Pos_Park_Vertical + gtyp_SSC.Vertical_Axis.Config.di_Pos_Window))
                   AND (gtyp_SSC.Vertical_Axis.di_Actual_Position >= (gtyp_SSC.di_Pos_Park_Vertical - gtyp_SSC.Vertical_Axis.Config.di_Pos_Window))
                   AND gtyp_SSC.Vertical_Axis.x_Position_Reached THEN
                   gtyp_SSC.Vertical_Axis.x_Start_Positioning := FALSE;
                   li_StepCase := 80;
               END_IF;

           80:
               gtyp_SSC.x_Park_Position_Reached := TRUE;



           ELSE
               ;
       END_CASE;

   ELSE
       lx_Init := TRUE;
   END_IF;
END_FUNCTION_BLOCK

FUNCTION_BLOCK PRG_SLD_Set_Counter_Values
   VAR
      lx_Init : Bool;
      lfb_R_Trig_Calib_activ : R_TRIG;
   END_VAR



   IF lx_Init THEN


       IF NOT gtyp_Setup.x_Counter_Value_Calibration THEN
           gtyp_Setup.i_Calib_CounterValue_Blue := gtyp_SLD.i_CounterValue_Blue;
           gtyp_Setup.i_Calib_CounterValue_Red := gtyp_SLD.i_CounterValue_Red;
           gtyp_Setup.i_Calib_CounterValue_White := gtyp_SLD.i_CounterValue_White;
       END_IF;


       IF gtyp_Setup.x_Set_CounterValues AND gtyp_Setup.x_Counter_Value_Calibration THEN
           gtyp_SLD.i_CounterValue_Blue := gtyp_Setup.i_Calib_CounterValue_Blue;
           gtyp_SLD.i_CounterValue_Red := gtyp_Setup.i_Calib_CounterValue_Red;
           gtyp_SLD.i_CounterValue_White := gtyp_Setup.i_Calib_CounterValue_White;
           gtyp_Setup.x_Set_CounterValues := FALSE;
       END_IF;

   ELSE
       lx_Init := TRUE;
   END_IF;
END_FUNCTION_BLOCK

FUNCTION_BLOCK PRG_VGR_Set_Park_Position
   VAR
      lx_Init : Bool;
      lx_Start_TON_Wait : Bool;
      lt_TON_Wait : Time;
      li_StepCase : Int;
      lfb_TON_Wait : TON_TIME;
      lfb_R_Trig_Start_Park_Pos : R_TRIG;
   END_VAR



   IF lx_Init THEN


       lfb_TON_Wait(IN := lx_Start_TON_Wait,
                     PT := lt_TON_Wait);

       lfb_R_Trig_Start_Park_Pos(CLK := gtyp_Setup.x_Park_Position
                                  OR IX_Set_Park_Position);


       IF lfb_R_Trig_Start_Park_Pos.Q THEN
           gtyp_VGR.x_Start_Park_Position := TRUE;
           li_StepCase := 0;
       END_IF;


       IF NOT gtyp_VGR.x_Start_Park_Position THEN
           li_StepCase := 0;
       END_IF;


       CASE li_StepCase OF

           0:
               lx_Start_TON_Wait := FALSE;
               li_StepCase := 10;

           10:
               IF gtyp_VGR.x_Start_Park_Position AND NOT gtyp_VGR.x_Park_Position_Reached THEN
                   gtyp_VGR.horizontal_Axis.x_Start_Positioning := FALSE;
                   gtyp_VGR.vertical_Axis.x_Start_Positioning := FALSE;
                   gtyp_VGR.rotate_Axis.x_Start_Positioning := FALSE;
                   gtyp_VGR.horizontal_Axis.x_Reference := FALSE;
                   gtyp_VGR.vertical_Axis.x_Reference := FALSE;
                   gtyp_VGR.rotate_Axis.x_Reference := FALSE;
                   gtyp_VGR.vertical_Axis.i_PWM := 800;
                   li_StepCase := 20;
               END_IF;

           20:
               gtyp_VGR.vertical_Axis.x_Reference := TRUE;

               IF NOT gtyp_VGR.vertical_Axis.x_Referenced THEN
                   li_StepCase := 30;
               END_IF;

           30:
               IF gtyp_VGR.vertical_Axis.x_Referenced THEN
                   gtyp_VGR.vertical_Axis.x_Reference := FALSE;
                   li_StepCase := 40;
               END_IF;

           40:
               gtyp_VGR.horizontal_Axis.x_Reference := TRUE;

               IF NOT gtyp_VGR.horizontal_Axis.x_Referenced THEN
                   li_StepCase := 50;
               END_IF;

           50:
               IF gtyp_VGR.horizontal_Axis.x_Referenced THEN
                   gtyp_VGR.horizontal_Axis.x_Reference := FALSE;
                   li_StepCase := 60;
               END_IF;

           60:
               gtyp_VGR.rotate_Axis.x_Reference := TRUE;

               IF NOT gtyp_VGR.rotate_Axis.x_Referenced THEN
                   li_StepCase := 70;
               END_IF;

           70:
               IF gtyp_VGR.rotate_Axis.x_Referenced THEN
                   gtyp_VGR.rotate_Axis.x_Reference := FALSE;
                   li_StepCase := 80;
               END_IF;

           80:
               gtyp_VGR.rotate_Axis.di_Target_Position   := gtyp_VGR.di_Pos_Park_rotate;
               gtyp_VGR.rotate_Axis.x_Start_Positioning  := TRUE;

               IF (gtyp_VGR.rotate_Axis.di_Actual_Position <= (gtyp_VGR.di_Pos_Park_rotate + gtyp_VGR.rotate_Axis.Config.di_Pos_Window))
                   AND (gtyp_VGR.rotate_Axis.di_Actual_Position >= (gtyp_VGR.di_Pos_Park_rotate - gtyp_VGR.rotate_Axis.Config.di_Pos_Window))
                   AND gtyp_VGR.rotate_Axis.x_Position_Reached THEN
                   gtyp_VGR.rotate_Axis.x_Start_Positioning := FALSE;
                   li_StepCase := 90;
               END_IF;

           90:
               gtyp_VGR.horizontal_Axis.di_Target_Position := gtyp_VGR.di_Pos_Park_horizontal;
               gtyp_VGR.horizontal_Axis.x_Start_Positioning := TRUE;

               IF (gtyp_VGR.horizontal_Axis.di_Actual_Position <= (gtyp_VGR.di_Pos_Park_horizontal + gtyp_VGR.horizontal_Axis.Config.di_Pos_Window))
                   AND (gtyp_VGR.horizontal_Axis.di_Actual_Position >= (gtyp_VGR.di_Pos_Park_horizontal - gtyp_VGR.horizontal_Axis.Config.di_Pos_Window))
                   AND gtyp_VGR.horizontal_Axis.x_Position_Reached THEN
                   gtyp_VGR.horizontal_Axis.x_Start_Positioning := FALSE;
                   li_StepCase := 100;
               END_IF;

           100:
               gtyp_VGR.vertical_Axis.i_PWM := 500;
               gtyp_VGR.vertical_Axis.di_Target_Position := gtyp_VGR.di_Pos_Park_vertical;
               gtyp_VGR.vertical_Axis.x_Start_Positioning := TRUE;

               IF (gtyp_VGR.vertical_Axis.di_Actual_Position <= (gtyp_VGR.di_Pos_Park_vertical + gtyp_VGR.vertical_Axis.Config.di_Pos_Window))
                   AND (gtyp_VGR.vertical_Axis.di_Actual_Position >= (gtyp_VGR.di_Pos_Park_vertical - gtyp_VGR.vertical_Axis.Config.di_Pos_Window))
                   AND gtyp_VGR.vertical_Axis.x_Position_Reached THEN
                   gtyp_VGR.vertical_Axis.x_Start_Positioning := FALSE;
                   li_StepCase := 110;
               END_IF;

           110:
               gtyp_VGR.x_Park_Position_Reached := TRUE;



           ELSE
               ;
       END_CASE;

   ELSE
       lx_Init := TRUE;
   END_IF;
END_FUNCTION_BLOCK

FUNCTION_BLOCK PRG_SSC_Axis_Horizontal
   VAR
      lx_Init : Bool;
      lfb_Horizontal_Axis : FB_Axis;
   END_VAR



   IF lx_Init THEN


       lfb_Horizontal_Axis(   ini_Axis                := 4,
                               indi_Increment          := gtyp_SSC.Horizontal_Axis.di_Increment,
                               inx_Ref_Switch          := IX_SSC_RefSwitchHorizontalAxis_I2,
                               inx_Referencing         := gtyp_SSC.Horizontal_Axis.x_Reference,
                               inx_Start_Positioning   := gtyp_SSC.Horizontal_Axis.x_Start_Positioning,
                               indi_Target_Position    := gtyp_SSC.Horizontal_Axis.di_Target_Position,
                               ini_PWM               := gtyp_SSC.Horizontal_Axis.i_PWM,
                               inouttyp_Config         := gtyp_SSC.Horizontal_Axis.Config,
                               inouttyp_Setup          := gtyp_SetupAxis);

       QX_SSC_M2_HorizontalAxisCounterclockwise_Q4      := lfb_Horizontal_Axis.outx_Motor_Neg;
       QX_SSC_M2_HorizontalAxisClockwise_Q3             := lfb_Horizontal_Axis.outx_Motor_Pos;
       QW_SSC_PWM_Horizontal_M2                         := lfb_Horizontal_Axis.outi_Motor_PWM;
       gtyp_SSC.Horizontal_Axis.di_Actual_Position   := lfb_Horizontal_Axis.outdi_Actual_Position;
       gtyp_SSC.Horizontal_Axis.x_Referenced         := lfb_Horizontal_Axis.outx_Referenced;
       gtyp_SSC.Horizontal_Axis.x_Position_Reached   := lfb_Horizontal_Axis.outx_Position_Reached;
   ELSE
       lx_Init := TRUE;
   END_IF;
END_FUNCTION_BLOCK

FUNCTION_BLOCK PRG_HBW_Set_Park_Position
   VAR
      lx_Init : Bool;
      lx_Start_TON_Wait : Bool;
      lt_TON_Wait : Time;
      li_StepCase : Int;
      lfb_TON_Wait : TON_TIME;
      lfb_R_Trig_Start_Park_Pos : R_TRIG;
   END_VAR



   IF lx_Init THEN


       lfb_TON_Wait(IN := lx_Start_TON_Wait,
                     PT := lt_TON_Wait);

       lfb_R_Trig_Start_Park_Pos(CLK := gtyp_Setup.x_Park_Position
                                  OR IX_Set_Park_Position);


       IF lfb_R_Trig_Start_Park_Pos.Q THEN
           gtyp_HBW.x_Start_Park_Position := TRUE;
           li_StepCase := 0;
       END_IF;


       IF NOT gtyp_HBW.x_Start_Park_Position THEN
           li_StepCase := 0;
       END_IF;


       CASE li_StepCase OF

           0:
               lx_Start_TON_Wait := FALSE;
               li_StepCase := 10;

           10:
               IF IX_HBW_SwitchCantileverFront_I5 OR NOT IX_HBW_SwitchCantileverBack_I6 THEN
                   QX_HBW_M4_CantileverBackward_Q8 := TRUE;
                   QX_HBW_M4_CantileverForward_Q7 := FALSE;
               ELSIF NOT IX_HBW_SwitchCantileverFront_I5 AND IX_HBW_SwitchCantileverBack_I6 THEN
                   QX_HBW_M4_CantileverBackward_Q8 := FALSE;
                   QX_HBW_M4_CantileverForward_Q7 := FALSE;
                   li_StepCase := 20;
               END_IF;

           20:
               IF gtyp_HBW.x_Start_Park_Position AND NOT gtyp_HBW.x_Park_Position_Reached THEN
                   gtyp_HBW.Horizontal_Axis.x_Start_Positioning := FALSE;
                   gtyp_HBW.Vertical_Axis.x_Start_Positioning := FALSE;
                   gtyp_HBW.Horizontal_Axis.x_Reference := FALSE;
                   gtyp_HBW.Vertical_Axis.x_Reference := FALSE;
                   QX_HBW_M4_CantileverBackward_Q8 := FALSE;
                   QX_HBW_M4_CantileverForward_Q7 := FALSE;
                   li_StepCase := 30;
               END_IF;

           30:
               gtyp_HBW.Vertical_Axis.x_Reference := TRUE;

               IF NOT gtyp_HBW.Vertical_Axis.x_Referenced THEN
                   li_StepCase := 40;
               END_IF;

           40:
               IF gtyp_HBW.Vertical_Axis.x_Referenced THEN
                   gtyp_HBW.Vertical_Axis.x_Reference := FALSE;
                   li_StepCase := 50;
               END_IF;

           50:
               gtyp_HBW.Horizontal_Axis.x_Reference := TRUE;

               IF NOT gtyp_HBW.Horizontal_Axis.x_Referenced THEN
                   li_StepCase := 60;
               END_IF;

           60:
               IF gtyp_HBW.Horizontal_Axis.x_Referenced THEN
                   gtyp_HBW.Horizontal_Axis.x_Reference := FALSE;
                   li_StepCase := 70;
               END_IF;

           70:
               gtyp_HBW.Horizontal_Axis.di_Target_Position := gtyp_HBW.di_Pos_Park_Horizontal;
               gtyp_HBW.Horizontal_Axis.x_Start_Positioning := TRUE;

               IF (gtyp_HBW.Horizontal_Axis.di_Actual_Position <= (gtyp_HBW.di_Pos_Park_Horizontal + gtyp_HBW.Horizontal_Axis.Config.di_Pos_Window))
                   AND (gtyp_HBW.Horizontal_Axis.di_Actual_Position >= (gtyp_HBW.di_Pos_Park_Horizontal - gtyp_HBW.Horizontal_Axis.Config.di_Pos_Window))
                   AND gtyp_HBW.Horizontal_Axis.x_Position_Reached THEN
                   gtyp_HBW.Horizontal_Axis.x_Start_Positioning := FALSE;
                   li_StepCase := 80;
               END_IF;

           80:
               gtyp_HBW.Vertical_Axis.di_Target_Position := gtyp_HBW.di_Pos_Park_Vertical;
               gtyp_HBW.Vertical_Axis.x_Start_Positioning := TRUE;

               IF (gtyp_HBW.Vertical_Axis.di_Actual_Position <= (gtyp_HBW.di_Pos_Park_Vertical + gtyp_HBW.Vertical_Axis.Config.di_Pos_Window))
                   AND (gtyp_HBW.Vertical_Axis.di_Actual_Position >= (gtyp_HBW.di_Pos_Park_Vertical - gtyp_HBW.Vertical_Axis.Config.di_Pos_Window))
                   AND gtyp_HBW.Vertical_Axis.x_Position_Reached THEN
                   gtyp_HBW.Vertical_Axis.x_Start_Positioning := FALSE;
                   li_StepCase := 90;
               END_IF;

           90:
               gtyp_HBW.x_Park_Position_Reached := TRUE;



           ELSE
               ;
       END_CASE;

   ELSE
       lx_Init := TRUE;
   END_IF;
END_FUNCTION_BLOCK

FUNCTION_BLOCK PRG_Acknowledge
   VAR
      lx_Init : Bool;
      li_StepCase : Int;
      lldt_Ack_old : LDT;
      lfb_TON_Wait : TON_TIME;
      lx_Start_TON_Wait : Bool;
   END_VAR



   IF lx_Init THEN
       lfb_TON_Wait(IN:= lx_Start_TON_Wait,PT:= T#20s);

       CASE li_StepCase OF

           0:
               lx_Start_TON_Wait := FALSE;


               IF (gtyp_Interface_Dashboard.Publish.ldt_AcknowledgeButton > lldt_Ack_old)
                   OR gtyp_Setup.x_AcknowledgeButton THEN
                   lldt_Ack_old    := gtyp_Interface_Dashboard.Publish.ldt_AcknowledgeButton;
                   li_StepCase    := 10;
               END_IF;

           10:
               gtyp_HBW.x_Error := FALSE;
               gtyp_MPO.x_Error := FALSE;
               gtyp_SLD.x_Error := FALSE;
               li_StepCase := 20;

           20:
               gtyp_Setup.x_AcknowledgeButton := FALSE;
               li_StepCase := 0;

       ELSE
           ;
       END_CASE;

   ELSE
       lx_Init := TRUE;
   END_IF;
END_FUNCTION_BLOCK

FUNCTION_BLOCK PRG_NFC
   VAR
      lx_Init : Bool;
      lx_Start : Bool;
      lx_Time_Wait : Bool;
      lx_Time_Error : Bool;
      li_StepCase : Int;
      ldt_MQTT : Date_And_Time;
      ldt_Delete_old : LDT;
      ldt_Read_old : LDT;
      li_Return_LDT : Int;
      lfb_TON_Error : TON_TIME;
      lfb_TON_Wait : TON_TIME;
   END_VAR



   IF lx_Init THEN


       lfb_TON_Error(IN:= lx_Time_Error,
                      PT:= T#30s);


       lfb_TON_Wait(IN := lx_Time_Wait,
                     PT := T#5s);


       CASE li_StepCase OF

           0:
               lx_Time_Wait                := FALSE;
               gtyp_VGR.x_NFC_Completed := FALSE;


               IF gtyp_VGR.x_NFC_Start_First AND NOT gtyp_VGR.x_Workpiece_NiO THEN
                   gtyp_Interface_TXT_Controler.Subscribe.State_NFC_Device.Workpiece.s_state := '';
                   gtyp_Interface_TXT_Controler.Subscribe.State_NFC_Device.Workpiece.s_type := '';

                   gtyp_Interface_TXT_Controler.Publish.ActionButtonNFCModule.s_cmd := '';
                   li_StepCase := 10;

               ELSIF gtyp_VGR.x_NFC_Start AND NOT gtyp_VGR.x_Workpiece_NiO THEN
                   gtyp_Interface_TXT_Controler.Publish.ActionButtonNFCModule.s_cmd := '';
                   li_StepCase := 40;

               ELSIF QX_SSC_LED_Green_Q5 AND NOT gtyp_VGR.x_Workpiece_NiO THEN
                   ldt_Read_old := gtyp_Interface_Dashboard.Publish.ActionButtonNFCModule.ldt_ts;
                   gtyp_VGR.x_NFC_Start_First := FALSE;
                   gtyp_VGR.x_NFC_Start := FALSE;
                   gtyp_Interface_TXT_Controler.Publish.ActionButtonNFCModule.s_cmd := '';
                   li_StepCase := 60;
               END_IF;

           10:

               gtyp_Interface_TXT_Controler.Publish.ActionButtonNFCModule.s_cmd := 'delete';
               li_Return_LDT := RD_SYS_T(ldt_MQTT);
               gtyp_Interface_TXT_Controler.Publish.ActionButtonNFCModule.ldt_ts := DT_TO_LDT(ldt_MQTT);

               li_StepCase := 20;

           20:
               lx_Time_Error := TRUE;
               IF (gtyp_Interface_TXT_Controler.Subscribe.State_NFC_Device.ldt_ts > gtyp_Interface_TXT_Controler.Publish.ActionButtonNFCModule.ldt_ts)
                   AND (gtyp_Interface_TXT_Controler.Subscribe.State_NFC_Device.Workpiece.s_type = 'NONE')
                   AND (gtyp_Interface_TXT_Controler.Subscribe.State_NFC_Device.Workpiece.s_state <> '')
                   AND (gtyp_Interface_TXT_Controler.Subscribe.State_NFC_Device.Workpiece.s_id <> '') THEN
                   gtyp_VGR.Workpiece.s_id := gtyp_Interface_TXT_Controler.Subscribe.State_NFC_Device.Workpiece.s_id;
                   lx_Time_Error := FALSE;
                   li_StepCase := 30;
               END_IF;

               IF lfb_TON_Error.Q THEN
                   lx_Time_Error := FALSE;
                   gtyp_VGR.x_Workpiece_NiO := TRUE;
                   li_StepCase := 0;
               END_IF;


           30:
               IF gtyp_Interface_TXT_Controler.Subscribe.State_NFC_Device.Workpiece.s_id <> '' THEN
                   li_StepCase := 40;
               END_IF;

           40:
               gtyp_Interface_TXT_Controler.Publish.ActionButtonNFCModule.History            := gtyp_VGR.History;
               gtyp_Interface_TXT_Controler.Publish.ActionButtonNFCModule.Workpiece.s_type   := gtyp_VGR.Workpiece.s_type;
               gtyp_Interface_TXT_Controler.Publish.ActionButtonNFCModule.Workpiece.s_state  := gtyp_VGR.Workpiece.s_state;

               li_Return_LDT := RD_SYS_T(ldt_MQTT);

               gtyp_Interface_TXT_Controler.Publish.ActionButtonNFCModule.s_cmd  := 'write';
               gtyp_Interface_TXT_Controler.Publish.ActionButtonNFCModule.ldt_ts := DT_TO_LDT(ldt_MQTT);

               li_StepCase := 50;

           50:
               lx_Time_Error := TRUE;
               IF (gtyp_Interface_TXT_Controler.Subscribe.State_NFC_Device.ldt_ts > gtyp_Interface_TXT_Controler.Publish.ActionButtonNFCModule.ldt_ts) THEN
                   lx_Time_Error := FALSE;
                   li_StepCase := 80;
               END_IF;

               IF lfb_TON_Error.Q THEN
                   lx_Time_Error := FALSE;
                   gtyp_VGR.x_Workpiece_NiO := TRUE;
                   li_StepCase := 0;
               END_IF;

           60:

               li_Return_LDT := RD_SYS_T(ldt_MQTT);

               gtyp_Interface_TXT_Controler.Publish.ActionButtonNFCModule.s_cmd := 'read_uid';
               gtyp_Interface_TXT_Controler.Publish.ActionButtonNFCModule.ldt_ts := DT_TO_LDT(ldt_MQTT);
               lx_Time_Wait   := TRUE;
               li_StepCase    := 70;

           70:
               IF NOT QX_SSC_LED_Green_Q5 OR lfb_TON_Wait.Q OR (gtyp_Interface_TXT_Controler.Subscribe.State_NFC_Device.ldt_ts > gtyp_Interface_TXT_Controler.Publish.ActionButtonNFCModule.ldt_ts) THEN
                   IF LEN(gtyp_Interface_TXT_Controler.Subscribe.State_NFC_Device.Workpiece.s_id) = 8 THEN
                       gtyp_Setup.x_Clean_Rack_HBW := TRUE;
                   END_IF;
                   lx_Time_Wait := FALSE;
                   gtyp_Interface_TXT_Controler.Subscribe.State_NFC_Device.Workpiece.s_id := '';
                   li_StepCase := 0;
               END_IF;

           80:

               gtyp_VGR.x_NFC_Completed := TRUE;

               IF NOT gtyp_VGR.x_NFC_Start AND NOT gtyp_VGR.x_NFC_Start_First THEN
                   gtyp_VGR.x_NFC_Completed := FALSE;
                   lx_Start := FALSE;
                   li_StepCase := 0;
               END_IF;


               ELSE
                   ;
       END_CASE;

   ELSE
       lx_Init := TRUE;
   END_IF;
END_FUNCTION_BLOCK

DATA_BLOCK PRG_VGR_Axis_vertical_DB

NON_RETAIN
PRG_VGR_Axis_vertical



END_DATA_BLOCK

DATA_BLOCK PRG_VGR_Ablauf_DB


NON_RETAIN
PRG_VGR_Ablauf



END_DATA_BLOCK

DATA_BLOCK PRG_VGR_Axis_horizontal_DB

NON_RETAIN
PRG_VGR_Axis_horizontal



END_DATA_BLOCK

DATA_BLOCK PRG_SSC_Axis_Vertical_DB


NON_RETAIN
PRG_SSC_Axis_Vertical



END_DATA_BLOCK

DATA_BLOCK PRG_SSC_Light_DB


NON_RETAIN
PRG_SSC_Light



END_DATA_BLOCK

DATA_BLOCK PRG_NFC_DB


NON_RETAIN
PRG_NFC



END_DATA_BLOCK

DATA_BLOCK PRG_SSC_Ablauf_DB


NON_RETAIN
PRG_SSC_Ablauf



END_DATA_BLOCK

DATA_BLOCK PRG_VGR_Axis_rotate_DB


NON_RETAIN
PRG_VGR_Axis_rotate



END_DATA_BLOCK

DATA_BLOCK RT_INFO_scl_OB30


NON_RETAIN
   VAR
      mode : UInt; obNbr : OB_ANY; infoData : LTime; returnValue : Int;
   END_VAR



   mode := 1;
   obNbr := 1;

END_DATA_BLOCK

DATA_BLOCK PRG_SSC_Axis_Horizontal_DB


NON_RETAIN
PRG_SSC_Axis_Horizontal



END_DATA_BLOCK

DATA_BLOCK PRG_SSC_Calibration_Color_DB


NON_RETAIN
PRG_SSC_Calibration_Color



END_DATA_BLOCK

DATA_BLOCK PRG_HBW_Axis_Vertical_DB


NON_RETAIN
PRG_HBW_Axis_Vertical



END_DATA_BLOCK

DATA_BLOCK PRG_SSC_Set_Positioning_DB


NON_RETAIN
PRG_SSC_Set_Positioning



END_DATA_BLOCK

DATA_BLOCK PRG_HBW_Set_Positioning_DB


NON_RETAIN
PRG_HBW_Set_Positioning



END_DATA_BLOCK

DATA_BLOCK PRG_VGR_Set_Positioning_DB


NON_RETAIN
PRG_VGR_Set_Positioning



END_DATA_BLOCK

DATA_BLOCK PRG_SLD_Calibration_Color_DB


NON_RETAIN
PRG_SLD_Calibration_Color



END_DATA_BLOCK

DATA_BLOCK PRG_SLD_Set_Counter_Values_DB


NON_RETAIN
PRG_SLD_Set_Counter_Values



END_DATA_BLOCK

DATA_BLOCK PRG_SSC_Set_Park_Position_DB
NON_RETAIN
PRG_SSC_Set_Park_Position



END_DATA_BLOCK

DATA_BLOCK PRG_VGR_Set_Park_Position_DB
NON_RETAIN
PRG_VGR_Set_Park_Position



END_DATA_BLOCK

DATA_BLOCK PRG_HBW_Set_Park_Position_DB
NON_RETAIN
PRG_HBW_Set_Park_Position



END_DATA_BLOCK

DATA_BLOCK RT_INFO_scl_OB1


NON_RETAIN
   VAR
      mode : UInt; obNbr : OB_ANY; infoData : LTime; returnValue : Int;
   END_VAR



   mode := 1;
   obNbr := 1;

END_DATA_BLOCK

DATA_BLOCK PRG_Acknowledge_DB


NON_RETAIN
PRG_Acknowledge



END_DATA_BLOCK

DATA_BLOCK PRG_DSO_Status_DB


NON_RETAIN
PRG_DSO_Status



END_DATA_BLOCK

DATA_BLOCK PRG_DSI_Status_DB


NON_RETAIN
PRG_DSI_Status



END_DATA_BLOCK

DATA_BLOCK PRG_Order_DB


NON_RETAIN
PRG_Order



END_DATA_BLOCK

DATA_BLOCK PRG_SLD_Ablauf_DB


NON_RETAIN
PRG_SLD_Ablauf



END_DATA_BLOCK

DATA_BLOCK PRG_MPO_Ablauf_DB


NON_RETAIN
PRG_MPO_Ablauf



END_DATA_BLOCK

DATA_BLOCK PRG_MPO_Set_Park_Position_DB
NON_RETAIN
PRG_MPO_Set_Park_Position



END_DATA_BLOCK

DATA_BLOCK PRG_HBW_Axis_Horizontal_DB


NON_RETAIN
PRG_HBW_Axis_Horizontal



END_DATA_BLOCK

DATA_BLOCK PRG_HBW_Ablauf_DB


NON_RETAIN
PRG_HBW_Ablauf



END_DATA_BLOCK

PROGRAM Main



   RT_INFO_scl_OB30.mode := 1;
   RT_INFO_scl_OB30.obNbr := 30;
   RT_INFO_scl_OB30.returnValue := RT_INFO(MODE := RT_INFO_scl_OB30.mode,
                                             OB := RT_INFO_scl_OB30.obNbr,
                                             INFO := RT_INFO_scl_OB30.infoData);


   RT_INFO_scl_OB1.mode := 1;
   RT_INFO_scl_OB1.obNbr := 1;
   RT_INFO_scl_OB1.returnValue := RT_INFO(MODE := RT_INFO_scl_OB1.mode,
                                            OB := RT_INFO_scl_OB1.obNbr,
                                            INFO := RT_INFO_scl_OB1.infoData);


   PRG_SSC_Ablauf_DB();
   PRG_SSC_Set_Positioning_DB();
   PRG_SSC_Set_Park_Position_DB();
   PRG_SSC_Calibration_Color_DB();
   PRG_SSC_Axis_Vertical_DB();
   PRG_SSC_Axis_Horizontal_DB();
   PRG_SSC_Light_DB();


   PRG_VGR_Ablauf_DB();
   PRG_VGR_Set_Positioning_DB();
   PRG_VGR_Set_Park_Position_DB();
   PRG_VGR_Axis_horizontal_DB();
   PRG_VGR_Axis_vertical_DB();
   PRG_VGR_Axis_rotate_DB();
   PRG_NFC_DB();


   PRG_HBW_Ablauf_DB();
   PRG_HBW_Set_Positioning_DB();
   PRG_HBW_Set_Park_Position_DB();
   PRG_HBW_Axis_Vertical_DB();
   PRG_HBW_Axis_Horizontal_DB();


   PRG_MPO_Ablauf_DB();
   PRG_MPO_Set_Park_Position_DB();


   PRG_SLD_Ablauf_DB();
   PRG_SLD_Calibration_Color_DB();
   PRG_SLD_Set_Counter_Values_DB();


   PRG_DSI_Status_DB();
   PRG_DSO_Status_DB();


   PRG_Order_DB();
   PRG_Acknowledge_DB();

END_PROGRAM
